INTERFACE ITcMessage_Ext

METHOD Send : BOOL
VAR_INPUT
	eventType : Tc3_EventLogger.TcEventEntry;
	args : STRING(255);
END_VAR
END_METHOD

END_INTERFACE

(* stored: Version 1.1.0.1, ProductVersion 3.1.4024.11
   Itf ITcMessage_Ext: Id {c659d345-17e7-4e7a-bcfb-ac2f396f1048}
   Method Send: Id {903682f6-fa6d-44e2-abfe-45550c59bb44} *)
